PROGRAM Simulation
VAR
	Idx					:	REAL;
	Level				: 	REAL;
END_VAR

VAR_OUTPUT
	LsLow: BOOL;
	LsMiddle: BOOL;
	LsHigh: BOOL;
END_VAR

Idx := Idx + 0.001;
Level := SIN(Idx);

Level := Level * 2000 + 2000;

LsLow 		:= Level >= 1500;
LsMiddle 	:= Level >= 2500;
LsHigh		:= NOT (Level >= 3500);

END_PROGRAM

(* stored: Version 1.1.0.1, ProductVersion 3.1.4024.15
   POU Simulation: Id {b069791d-3638-4eb3-9379-9d80a282a7a0}, SpecialFunc None *)
